# EPICS autosave request: apps/myaDataApp/Db/harpScanDataAll.req
file harpScanData.req P=HB_BEAM:SCAN:,R=tagger:
file harpScanData.req P=HB_BEAM:SCAN:,R=2H02A:
